// TIA Portal V20 export
TYPE "TypeHeaderPcGld"
   STRUCT
      valid : Int;   // valid
      watchdog : Int;   // watchdog
      bit40 : Bool;
      ack : Bool;   // acknowledge
      bit42 : Bool;
      bit43 : Bool;
      bit44 : Bool;
      bit45 : Bool;
      bit46 : Bool;
      bit47 : Bool;
      word6 : Word;
      word8 : Word;
   END_STRUCT;
END_TYPE
